// TwinCAT 3 PLC project Untitled1
// ProgramVersion: 3.1.4026.11
// libraries:
//   Tc2_Standard, * (Beckhoff Automation GmbH)
//   Tc2_System, * (Beckhoff Automation GmbH)
// project tree:
//   / PlcTask.TcTTO
//   POUs/ MAIN.TcPOU, FB_Counter.TcPOU, FB_CustomTimer.TcPOU, FB_StateMachine.TcPOU, FB_TestRunner.TcPOU
//   DUTs/ E_MachineState.TcDUT, ST_TestResults.TcDUT
// real-time tasks:
//   TASK PlcTask: cycle T#10ms, priority 20, ADS port 350

CONFIGURATION Untitled1
    RESOURCE PLC ON TwinCAT3
        TASK PlcTask(INTERVAL := T#10ms, PRIORITY := 20);
        PROGRAM MAIN WITH PlcTask : MAIN;
    END_RESOURCE
END_CONFIGURATION

// ---- DUTs/E_MachineState.TcDUT
{attribute 'qualified_only'}
{attribute 'strict'}
TYPE E_MachineState :
(
    Idle        := 0,   // Machine is idle
    Starting    := 1,   // Machine is starting
    Running     := 2,   // Machine is running
    Paused      := 3,   // Machine is paused
    Stopping    := 4,   // Machine is stopping
    Error       := 5,   // Error state
    Emergency   := 6    // Emergency stop
) := Idle;
END_TYPE

// ---- DUTs/ST_TestResults.TcDUT
TYPE ST_TestResults :
STRUCT
    // Test counters
    iTestsTotal     : INT;      // Total number of tests
    iTestsPassed    : INT;      // Number of passed tests
    iTestsFailed    : INT;      // Number of failed tests

    // Current test info
    sCurrentTest    : STRING;   // Current test name
    bTestRunning    : BOOL;     // Test is running
    bAllTestsPassed : BOOL;     // All tests passed flag

    // Individual test results
    bCounterTest    : BOOL;     // Counter FB test result
    bTimerTest      : BOOL;     // Timer FB test result
    bStateMachineTest : BOOL;   // State machine FB test result

    // Error messages
    sLastError      : STRING;   // Last error message
END_STRUCT
END_TYPE

// ---- POUs/MAIN.TcPOU
PROGRAM MAIN
VAR
    // Test mode selection
    bAutoTest       : BOOL := TRUE;     // Run automated tests
    bManualTest     : BOOL := FALSE;    // Run manual tests

    // Automated test runner
    fbTestRunner    : FB_TestRunner;
    bRunTests       : BOOL;             // Trigger to start tests
    bResetTests     : BOOL;             // Reset test results

    // Manual test instances
    fbCounter       : FB_Counter;
    fbTimer         : FB_CustomTimer;
    fbStateMachine  : FB_StateMachine;

    // Manual test controls
    bCounterEnable  : BOOL;
    bCountUp        : BOOL;
    bCountDown      : BOOL;
    bTimerStart     : BOOL;
    bTimerReset     : BOOL;
    bMachineStart   : BOOL;
    bMachineStop    : BOOL;
    bMachinePause   : BOOL;
    bMachineReset   : BOOL;
END_VAR

//==============================================================================
// FB Test Program - MAIN
// Description: Tests all generated Function Blocks
// Mode: Auto (automated tests) or Manual (interactive testing)
//==============================================================================

IF bAutoTest THEN
    //--------------------------------------------------------------------------
    // AUTOMATED TESTING MODE
    //--------------------------------------------------------------------------
    // Run the automated test suite
    fbTestRunner(
        bRunTests := bRunTests,
        bResetTests := bResetTests
    );

    // Display test results in watch window:
    // fbTestRunner.stResults.sCurrentTest
    // fbTestRunner.stResults.iTestsPassed
    // fbTestRunner.stResults.iTestsFailed
    // fbTestRunner.stResults.bAllTestsPassed

ELSIF bManualTest THEN
    //--------------------------------------------------------------------------
    // MANUAL TESTING MODE
    //--------------------------------------------------------------------------

    // Test Counter FB
    fbCounter(
        bEnable := bCounterEnable,
        bReset := FALSE,
        bCountUp := bCountUp,
        bCountDown := bCountDown,
        iMin := 0,
        iMax := 100
    );

    // Test Timer FB
    fbTimer(
        bStart := bTimerStart,
        bStop := FALSE,
        bReset := bTimerReset,
        tSetTime := T#5S
    );

    // Test State Machine FB
    fbStateMachine(
        bStart := bMachineStart,
        bStop := bMachineStop,
        bPause := bMachinePause,
        bReset := bMachineReset,
        bEmergency := FALSE
    );

    // Watch these variables to see the results:
    // fbCounter.iCount, fbCounter.bMaxReached, fbCounter.bMinReached
    // fbTimer.tElapsed, fbTimer.rProgress, fbTimer.bDone
    // fbStateMachine.eState, fbStateMachine.sStateText, fbStateMachine.iCycles
END_IF

END_PROGRAM

// ---- POUs/FB_TestRunner.TcPOU
FUNCTION_BLOCK FB_TestRunner
VAR_INPUT
    bRunTests   : BOOL;     // Start running all tests
    bResetTests : BOOL;     // Reset test results
END_VAR

VAR_OUTPUT
    stResults   : ST_TestResults; // Test results
END_VAR

VAR
    // Test state machine
    eTestState  : (INIT, TEST_COUNTER, TEST_TIMER, TEST_STATEMACHINE, COMPLETE);
    iTestStep   : INT;
    fbTestTimer : TON;

    // FB instances for testing
    fbCounter   : FB_Counter;
    fbTimer     : FB_CustomTimer;
    fbStateMachine : FB_StateMachine;

    // Test variables
    iCycleCount : INT;
    bTestFlag   : BOOL;
END_VAR

// Reset tests
IF bResetTests THEN
    eTestState := INIT;
    iTestStep := 0;
    stResults.iTestsTotal := 0;
    stResults.iTestsPassed := 0;
    stResults.iTestsFailed := 0;
    stResults.bTestRunning := FALSE;
    stResults.bAllTestsPassed := FALSE;
    stResults.bCounterTest := FALSE;
    stResults.bTimerTest := FALSE;
    stResults.bStateMachineTest := FALSE;
    stResults.sCurrentTest := '';
    stResults.sLastError := '';
    iCycleCount := 0;
    RETURN;
END_IF

// Run tests when triggered
IF NOT bRunTests THEN
    RETURN;
END_IF

stResults.bTestRunning := TRUE;

// Test state machine
CASE eTestState OF
    INIT:
        stResults.iTestsTotal := 3;
        stResults.sCurrentTest := 'Initializing tests...';
        iTestStep := 0;
        eTestState := TEST_COUNTER;

    TEST_COUNTER:
        stResults.sCurrentTest := 'Testing Counter FB';

        CASE iTestStep OF
            0: // Reset counter
                fbCounter(bReset := TRUE);
                IF fbCounter.iCount = 0 THEN
                    iTestStep := 1;
                END_IF

            1: // Enable and count up
                fbCounter(bEnable := TRUE, bReset := FALSE, bCountUp := TRUE, bCountDown := FALSE, iMax := 10);
                iCycleCount := iCycleCount + 1;
                IF iCycleCount > 5 THEN
                    IF fbCounter.iCount >= 5 THEN
                        iTestStep := 2;
                        iCycleCount := 0;
                    ELSE
                        stResults.sLastError := 'Counter: Count up failed';
                        stResults.iTestsFailed := stResults.iTestsFailed + 1;
                        eTestState := TEST_TIMER;
                        iTestStep := 0;
                    END_IF
                END_IF

            2: // Count down
                fbCounter(bEnable := TRUE, bCountUp := FALSE, bCountDown := TRUE);
                iCycleCount := iCycleCount + 1;
                IF iCycleCount > 5 THEN
                    IF fbCounter.iCount < 5 THEN
                        stResults.bCounterTest := TRUE;
                        stResults.iTestsPassed := stResults.iTestsPassed + 1;
                        eTestState := TEST_TIMER;
                        iTestStep := 0;
                        iCycleCount := 0;
                    ELSE
                        stResults.sLastError := 'Counter: Count down failed';
                        stResults.iTestsFailed := stResults.iTestsFailed + 1;
                        eTestState := TEST_TIMER;
                        iTestStep := 0;
                    END_IF
                END_IF
        END_CASE

    TEST_TIMER:
        stResults.sCurrentTest := 'Testing Timer FB';

        CASE iTestStep OF
            0: // Reset timer
                fbTimer(bReset := TRUE);
                IF NOT fbTimer.bRunning AND NOT fbTimer.bDone THEN
                    iTestStep := 1;
                END_IF

            1: // Start timer
                fbTimer(bStart := TRUE, bReset := FALSE, tSetTime := T#500MS);
                IF fbTimer.bRunning THEN
                    iTestStep := 2;
                    iCycleCount := 0;
                END_IF

            2: // Wait for completion
                fbTimer(bStart := FALSE);
                iCycleCount := iCycleCount + 1;

                // Timeout after 100 cycles (1 second at 10ms cycle)
                IF fbTimer.bDone OR iCycleCount > 100 THEN
                    IF fbTimer.bDone AND fbTimer.rProgress >= 99.0 THEN
                        stResults.bTimerTest := TRUE;
                        stResults.iTestsPassed := stResults.iTestsPassed + 1;
                    ELSE
                        stResults.sLastError := 'Timer: Did not complete in time';
                        stResults.iTestsFailed := stResults.iTestsFailed + 1;
                    END_IF
                    eTestState := TEST_STATEMACHINE;
                    iTestStep := 0;
                    iCycleCount := 0;
                END_IF
        END_CASE

    TEST_STATEMACHINE:
        stResults.sCurrentTest := 'Testing State Machine FB';

        CASE iTestStep OF
            0: // Initial state should be Idle
                fbStateMachine(bStart := FALSE, bStop := FALSE, bReset := FALSE);
                IF fbStateMachine.eState = E_MachineState.Idle THEN
                    iTestStep := 1;
                END_IF

            1: // Start machine
                fbStateMachine(bStart := TRUE);
                iCycleCount := iCycleCount + 1;
                IF fbStateMachine.eState = E_MachineState.Starting OR iCycleCount > 10 THEN
                    iTestStep := 2;
                    iCycleCount := 0;
                END_IF

            2: // Wait for running state
                fbStateMachine(bStart := FALSE);
                iCycleCount := iCycleCount + 1;
                IF fbStateMachine.eState = E_MachineState.Running OR iCycleCount > 250 THEN
                    IF fbStateMachine.eState = E_MachineState.Running THEN
                        iTestStep := 3;
                    ELSE
                        stResults.sLastError := 'StateMachine: Did not reach Running state';
                        stResults.iTestsFailed := stResults.iTestsFailed + 1;
                        eTestState := COMPLETE;
                    END_IF
                    iCycleCount := 0;
                END_IF

            3: // Stop machine
                fbStateMachine(bStop := TRUE);
                iCycleCount := iCycleCount + 1;
                IF fbStateMachine.eState = E_MachineState.Stopping OR iCycleCount > 10 THEN
                    iTestStep := 4;
                    iCycleCount := 0;
                END_IF

            4: // Wait for idle state
                fbStateMachine(bStop := FALSE);
                iCycleCount := iCycleCount + 1;
                IF fbStateMachine.eState = E_MachineState.Idle OR iCycleCount > 150 THEN
                    IF fbStateMachine.eState = E_MachineState.Idle THEN
                        stResults.bStateMachineTest := TRUE;
                        stResults.iTestsPassed := stResults.iTestsPassed + 1;
                    ELSE
                        stResults.sLastError := 'StateMachine: Did not return to Idle';
                        stResults.iTestsFailed := stResults.iTestsFailed + 1;
                    END_IF
                    eTestState := COMPLETE;
                    iCycleCount := 0;
                END_IF
        END_CASE

    COMPLETE:
        stResults.sCurrentTest := 'Tests Complete';
        stResults.bTestRunning := FALSE;
        stResults.bAllTestsPassed := (stResults.iTestsFailed = 0) AND (stResults.iTestsPassed = stResults.iTestsTotal);
END_CASE

END_FUNCTION_BLOCK

// ---- POUs/FB_Counter.TcPOU
FUNCTION_BLOCK FB_Counter
VAR_INPUT
    bEnable     : BOOL;     // Enable counter
    bReset      : BOOL;     // Reset counter to 0
    bCountUp    : BOOL;     // Count up trigger
    bCountDown  : BOOL;     // Count down trigger
    iMin        : INT := 0; // Minimum value
    iMax        : INT := 100; // Maximum value
END_VAR

VAR_OUTPUT
    iCount      : INT;      // Current count value
    bMinReached : BOOL;     // TRUE when min value reached
    bMaxReached : BOOL;     // TRUE when max value reached
    bError      : BOOL;     // Error flag
    sErrorMsg   : STRING;   // Error message
END_VAR

VAR
    bCountUpOld   : BOOL;   // Previous state of count up
    bCountDownOld : BOOL;   // Previous state of count down
END_VAR

// Reset counter
IF bReset THEN
    iCount := 0;
    bError := FALSE;
    sErrorMsg := '';
    bMinReached := FALSE;
    bMaxReached := FALSE;
    bCountUpOld := FALSE;
    bCountDownOld := FALSE;
    RETURN;
END_IF

// Check for valid range
IF iMin > iMax THEN
    bError := TRUE;
    sErrorMsg := 'Error: Min > Max';
    RETURN;
END_IF

// Counter logic when enabled
IF bEnable THEN
    // Count up on rising edge
    IF bCountUp AND NOT bCountUpOld THEN
        IF iCount < iMax THEN
            iCount := iCount + 1;
        ELSE
            bMaxReached := TRUE;
        END_IF
    END_IF

    // Count down on rising edge
    IF bCountDown AND NOT bCountDownOld THEN
        IF iCount > iMin THEN
            iCount := iCount - 1;
        ELSE
            bMinReached := TRUE;
        END_IF
    END_IF

    // Update boundary flags
    bMinReached := (iCount <= iMin);
    bMaxReached := (iCount >= iMax);
ELSE
    // Disabled - maintain current value
END_IF

// Store previous states
bCountUpOld := bCountUp;
bCountDownOld := bCountDown;

END_FUNCTION_BLOCK

// ---- POUs/FB_CustomTimer.TcPOU
FUNCTION_BLOCK FB_CustomTimer
VAR_INPUT
    bStart      : BOOL;         // Start timer
    bStop       : BOOL;         // Stop timer
    bReset      : BOOL;         // Reset timer
    tSetTime    : TIME := T#1S; // Set time duration
END_VAR

VAR_OUTPUT
    bRunning    : BOOL;         // Timer is running
    bDone       : BOOL;         // Timer completed
    tElapsed    : TIME;         // Elapsed time
    tRemaining  : TIME;         // Remaining time
    rProgress   : REAL;         // Progress percentage (0-100)
END_VAR

VAR
    tStartTime  : TIME;         // Start timestamp
    fbTON       : TON;          // Internal TON timer
END_VAR

// Reset timer
IF bReset THEN
    bRunning := FALSE;
    bDone := FALSE;
    tElapsed := T#0S;
    tRemaining := tSetTime;
    rProgress := 0.0;
    fbTON(IN := FALSE);
    RETURN;
END_IF

// Stop timer
IF bStop THEN
    bRunning := FALSE;
    fbTON(IN := FALSE);
    RETURN;
END_IF

// Start timer
IF bStart AND NOT bRunning THEN
    bRunning := TRUE;
    bDone := FALSE;
    tElapsed := T#0S;
    rProgress := 0.0;
END_IF

// Timer logic
IF bRunning THEN
    fbTON(IN := TRUE, PT := tSetTime);

    tElapsed := fbTON.ET;
    tRemaining := tSetTime - tElapsed;

    // Calculate progress percentage
    IF TIME_TO_DWORD(tSetTime) > 0 THEN
        rProgress := (TIME_TO_DWORD(tElapsed) * 100.0) / TIME_TO_DWORD(tSetTime);
    END_IF

    // Check if done
    IF fbTON.Q THEN
        bDone := TRUE;
        bRunning := FALSE;
        rProgress := 100.0;
        tRemaining := T#0S;
    END_IF
ELSE
    fbTON(IN := FALSE);
END_IF

END_FUNCTION_BLOCK

// ---- POUs/FB_StateMachine.TcPOU
FUNCTION_BLOCK FB_StateMachine
VAR_INPUT
    bStart      : BOOL;     // Start command
    bStop       : BOOL;     // Stop command
    bReset      : BOOL;     // Reset command
    bPause      : BOOL;     // Pause command
    bEmergency  : BOOL;     // Emergency stop
END_VAR

VAR_OUTPUT
    eState      : E_MachineState; // Current state
    bBusy       : BOOL;     // Machine is busy
    bError      : BOOL;     // Error occurred
    sStateText  : STRING;   // State description
    iCycles     : INT;      // Cycle counter
END_VAR

VAR
    eLastState  : E_MachineState;
    fbTimer     : TON;
END_VAR

// Emergency stop - highest priority
IF bEmergency THEN
    eState := E_MachineState.Emergency;
    bError := TRUE;
    bBusy := FALSE;
    sStateText := 'EMERGENCY STOP';
    RETURN;
END_IF

// State machine logic
CASE eState OF
    E_MachineState.Idle:
        bBusy := FALSE;
        bError := FALSE;
        sStateText := 'Idle - Ready to start';

        IF bStart THEN
            eState := E_MachineState.Starting;
        END_IF

    E_MachineState.Starting:
        bBusy := TRUE;
        sStateText := 'Starting...';

        // Simulate startup time
        fbTimer(IN := TRUE, PT := T#2S);
        IF fbTimer.Q THEN
            fbTimer(IN := FALSE);
            eState := E_MachineState.Running;
            iCycles := 0;
        END_IF

        IF bStop THEN
            fbTimer(IN := FALSE);
            eState := E_MachineState.Stopping;
        END_IF

    E_MachineState.Running:
        bBusy := TRUE;
        sStateText := 'Running';
        iCycles := iCycles + 1;

        IF bStop THEN
            eState := E_MachineState.Stopping;
        ELSIF bPause THEN
            eState := E_MachineState.Paused;
        END_IF

    E_MachineState.Paused:
        bBusy := TRUE;
        sStateText := 'Paused';

        IF bStart THEN
            eState := E_MachineState.Running;
        ELSIF bStop THEN
            eState := E_MachineState.Stopping;
        END_IF

    E_MachineState.Stopping:
        bBusy := TRUE;
        sStateText := 'Stopping...';

        // Simulate shutdown time
        fbTimer(IN := TRUE, PT := T#1S);
        IF fbTimer.Q THEN
            fbTimer(IN := FALSE);
            eState := E_MachineState.Idle;
        END_IF

    E_MachineState.Emergency:
        bBusy := FALSE;
        bError := TRUE;
        sStateText := 'EMERGENCY - Reset required';

        IF bReset AND NOT bEmergency THEN
            bError := FALSE;
            eState := E_MachineState.Idle;
        END_IF

    E_MachineState.Error:
        bBusy := FALSE;
        bError := TRUE;
        sStateText := 'Error - Reset required';

        IF bReset THEN
            bError := FALSE;
            eState := E_MachineState.Idle;
        END_IF
END_CASE

// Reset command
IF bReset AND NOT bEmergency THEN
    IF eState = E_MachineState.Error OR eState = E_MachineState.Emergency THEN
        eState := E_MachineState.Idle;
        bError := FALSE;
    END_IF
END_IF

END_FUNCTION_BLOCK
